// TIA Portal V16 export
// export: Created 2025-05-24T14:53:42.6954034Z, ExportSetting WithDefaults, DisplayName Totally Integrated Automation Portal, DisplayVersion V16, DisplayName TIA Portal Version Control Interface, DisplayVersion V16, DisplayName TIA Portal Openness, DisplayVersion V16, DisplayName STEP 7 Professional, DisplayVersion V16, DisplayName STEP 7 Safety, DisplayVersion V16, DisplayName WinCC Advanced, DisplayVersion V16
ORGANIZATION_BLOCK "OB1"   // OB1, LAD, ProgramCycle
TITLE = MAIN Program
VERSION : 0.1
// MAIN Block
// stored: IsIECCheckEnabled false
   VAR_TEMP
      Temp_0 : Byte;
      Temp_1 : Byte;
      Temp_2 : Byte;
      Temp_3 : Byte;
      Temp_4 : Byte;
      Temp_5 : Byte;
      Temp_6 : Int;
      Temp_7 : Int;
      Temp_8 : Int;
      Temp_9 : Date_And_Time;
      Temp_10 : DWord;
      EncoderDirection : Bool;
      HomingActive : Bool;
      EncError : Bool;
      SafetyActive : Bool;
      "Spare Drive 6" : Bool;
      "Spare Drive 7" : Bool;
      "Spare Drive 8" : Bool;
      "Spare Drive 9" : Bool;
      "Spare Drive 10" : Bool;
      SAFE_OK_Signal : Bool;
      Raw_Position : Real;
      Encoder : Int;
      Gate : Bool;
      GATESTP : Bool;
      OTERRA : Bool;
      Direct : Bool;
      Prepar : Bool;
      CMPV1 : Bool;
      CMPV2 : Bool;
      RESSYNC : Bool;
      RESZERO : Bool;
      OTERR : Bool;
      UnscPos : Int;
      Sc_Pos : Int;
      ActEncPos : Real;
      Start_ReferenceRun : Bool;
      ReferenceSwitch_Input : Bool;
      "Reference Position" : Real;
      "Jog FWD" : Bool;
      "Jog REV" : Bool;
      RefSwitchTemp : Bool;
      RefPosDint : DInt;
      RefPosInt : Real;
      Start_Movement : Bool;
      ClockTime : Int;
      LT_Time : Date_And_Time;
      Summer : Bool;
      SystemStartUp : Bool;
      StartupLow : Bool;
      ManualSensorOverride : Bool;
      Axis1_ScaledPosition : Real;
      Axis1_ActualEncPosition : Real;
   END_VAR
   VAR_TEMP   // added for the SCL form of the ladder/FBD networks
      _w1 : Bool;
   END_VAR
BEGIN

REGION Network 1: Retain Variables
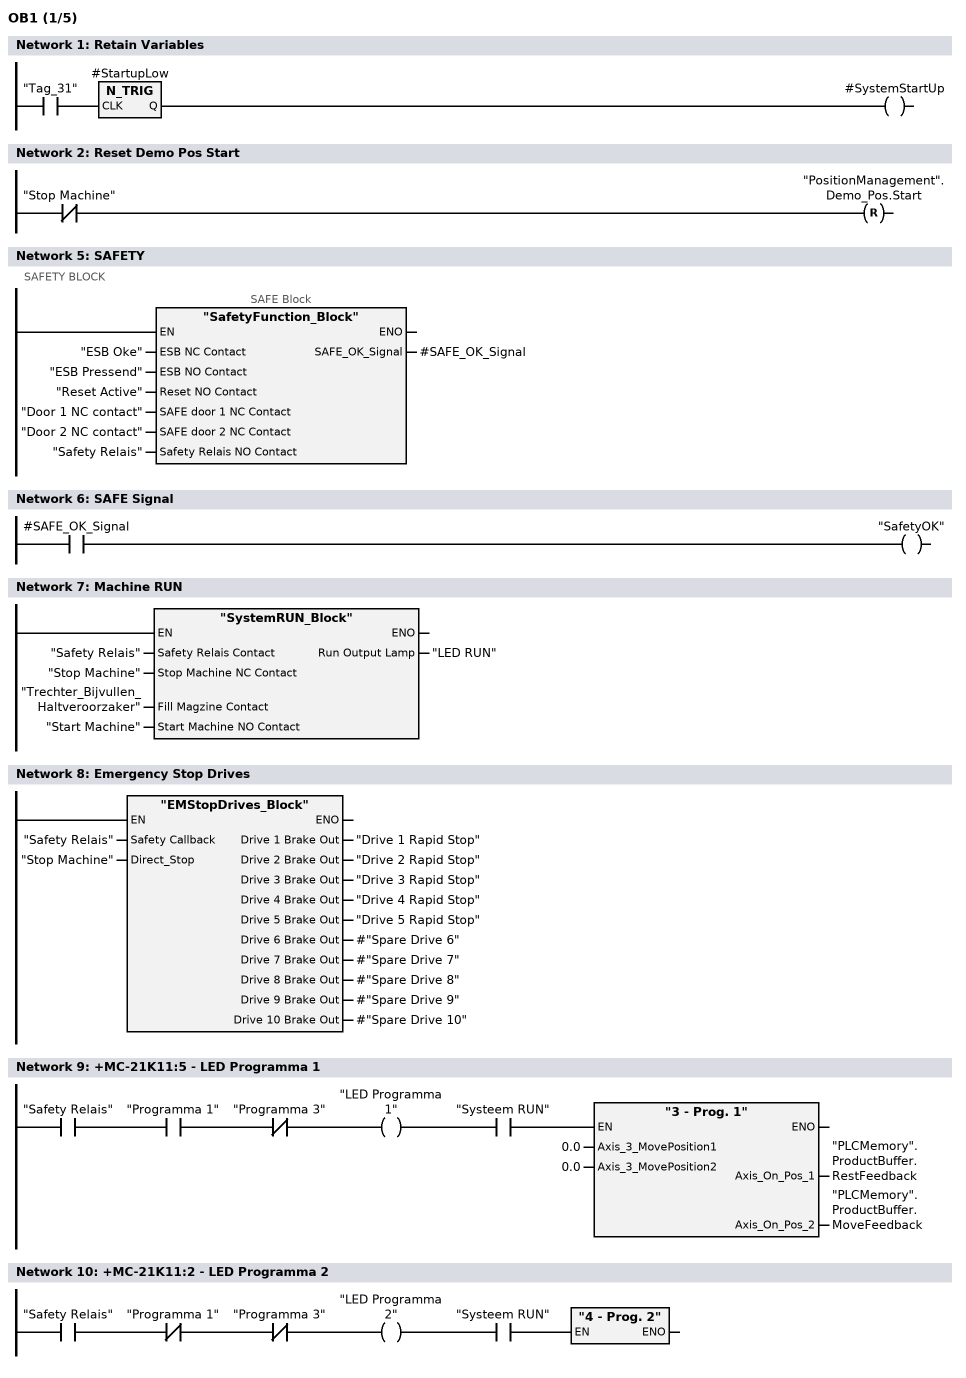
   RUNG wire#powerrail
      Contact( "Tag_31" )
      N_Trig( #StartupLow )
      Coil( #SystemStartUp )
   END_RUNG
   // the same network as SCL:
   #_w1 := NOT "Tag_31" AND #StartupLow;   // falling edge
   #StartupLow := "Tag_31";
   #SystemStartUp := #_w1;
END_REGION

REGION Network 2: Reset Demo Pos Start
   RUNG wire#powerrail
      I_Contact( "Stop Machine" )
      R_Coil( "PositionManagement".Demo_Pos.Start )
   END_RUNG
   // the same network as SCL:
   IF NOT "Stop Machine" THEN "PositionManagement".Demo_Pos.Start := FALSE; END_IF;
END_REGION

REGION Network 3: Retain Veriables (2)
END_REGION

REGION Network 4: System Time
END_REGION

REGION Network 5: SAFETY
   // SAFETY BLOCK
   RUNG wire#powerrail
      "SafetyFunction_Block"("ESB NC Contact" := "ESB Oke", "ESB NO Contact" := "ESB Pressend", "Reset NO Contact" := "Reset Active", "SAFE door 1 NC Contact" := "Door 1 NC contact", "SAFE door 2 NC Contact" := "Door 2 NC contact", "Safety Relais NO Contact" := "Safety Relais", SAFE_OK_Signal => #SAFE_OK_Signal)   // SAFE Block
   END_RUNG
   // the same network as SCL:
   "SafetyFunction_Block"("ESB NC Contact" := "ESB Oke",   // SAFE Block
                          "ESB NO Contact" := "ESB Pressend",
                          "Reset NO Contact" := "Reset Active",
                          "SAFE door 1 NC Contact" := "Door 1 NC contact",
                          "SAFE door 2 NC Contact" := "Door 2 NC contact",
                          "Safety Relais NO Contact" := "Safety Relais",
                          SAFE_OK_Signal => #SAFE_OK_Signal);
END_REGION

REGION Network 6: SAFE Signal
   RUNG wire#powerrail
      Contact( #SAFE_OK_Signal )
      Coil( "SafetyOK" )
   END_RUNG
   // the same network as SCL:
   "SafetyOK" := #SAFE_OK_Signal;
END_REGION

REGION Network 7: Machine RUN
   RUNG wire#powerrail
      "SystemRUN_Block"("Safety Relais Contact" := "Safety Relais", "Stop Machine NC Contact" := "Stop Machine", "Fill Magzine Contact" := "Trechter_Bijvullen_Haltveroorzaker", "Start Machine NO Contact" := "Start Machine", "Run Output Lamp" => "LED RUN")
   END_RUNG
   // the same network as SCL:
   "SystemRUN_Block"("Safety Relais Contact" := "Safety Relais",
                     "Stop Machine NC Contact" := "Stop Machine",
                     "Fill Magzine Contact" := "Trechter_Bijvullen_Haltveroorzaker",
                     "Start Machine NO Contact" := "Start Machine",
                     "Run Output Lamp" => "LED RUN");
END_REGION

REGION Network 8: Emergency Stop Drives
   RUNG wire#powerrail
      "EMStopDrives_Block"("Safety Callback" := "Safety Relais", Direct_Stop := "Stop Machine", "Drive 1 Brake Out" => "Drive 1 Rapid Stop", "Drive 2 Brake Out" => "Drive 2 Rapid Stop", "Drive 3 Brake Out" => "Drive 3 Rapid Stop", "Drive 4 Brake Out" => "Drive 4 Rapid Stop", "Drive 5 Brake Out" => "Drive 5 Rapid Stop", "Drive 6 Brake Out" => #"Spare Drive 6", "Drive 7 Brake Out" => #"Spare Drive 7", "Drive 8 Brake Out" => #"Spare Drive 8", "Drive 9 Brake Out" => #"Spare Drive 9", "Drive 10 Brake Out" => #"Spare Drive 10")
   END_RUNG
   // the same network as SCL:
   "EMStopDrives_Block"("Safety Callback" := "Safety Relais",
                        Direct_Stop := "Stop Machine",
                        "Drive 1 Brake Out" => "Drive 1 Rapid Stop",
                        "Drive 2 Brake Out" => "Drive 2 Rapid Stop",
                        "Drive 3 Brake Out" => "Drive 3 Rapid Stop",
                        "Drive 4 Brake Out" => "Drive 4 Rapid Stop",
                        "Drive 5 Brake Out" => "Drive 5 Rapid Stop",
                        "Drive 6 Brake Out" => #"Spare Drive 6",
                        "Drive 7 Brake Out" => #"Spare Drive 7",
                        "Drive 8 Brake Out" => #"Spare Drive 8",
                        "Drive 9 Brake Out" => #"Spare Drive 9",
                        "Drive 10 Brake Out" => #"Spare Drive 10");
END_REGION

REGION Network 9: +MC-21K11:5 - LED Programma 1
   RUNG wire#powerrail
      Contact( "Safety Relais" )
      Contact( "Programma 1" )
      I_Contact( "Programma 3" )
      Coil( "LED Programma 1" )
      Contact( "Systeem RUN" )
      "3 - Prog. 1"(Axis_3_MovePosition1 := 0.0, Axis_3_MovePosition2 := 0.0, Axis_On_Pos_1 => "PLCMemory".ProductBuffer.RestFeedback, Axis_On_Pos_2 => "PLCMemory".ProductBuffer.MoveFeedback)
   END_RUNG
   // the same network as SCL:
   "LED Programma 1" := "Safety Relais" AND "Programma 1" AND NOT "Programma 3";
   IF "LED Programma 1" AND "Systeem RUN" THEN
       "3 - Prog. 1"(Axis_3_MovePosition1 := 0.0,
                     Axis_3_MovePosition2 := 0.0,
                     Axis_On_Pos_1 => "PLCMemory".ProductBuffer.RestFeedback,
                     Axis_On_Pos_2 => "PLCMemory".ProductBuffer.MoveFeedback);
   END_IF;
END_REGION

REGION Network 10: +MC-21K11:2 - LED Programma 2
   RUNG wire#powerrail
      Contact( "Safety Relais" )
      I_Contact( "Programma 1" )
      I_Contact( "Programma 3" )
      Coil( "LED Programma 2" )
      Contact( "Systeem RUN" )
      "4 - Prog. 2"()
   END_RUNG
   // the same network as SCL:
   "LED Programma 2" := "Safety Relais" AND NOT "Programma 1" AND NOT "Programma 3";
   IF "LED Programma 2" AND "Systeem RUN" THEN "4 - Prog. 2"(); END_IF;
END_REGION

REGION Network 11: +MC-21K11:6 - LED Programma 3
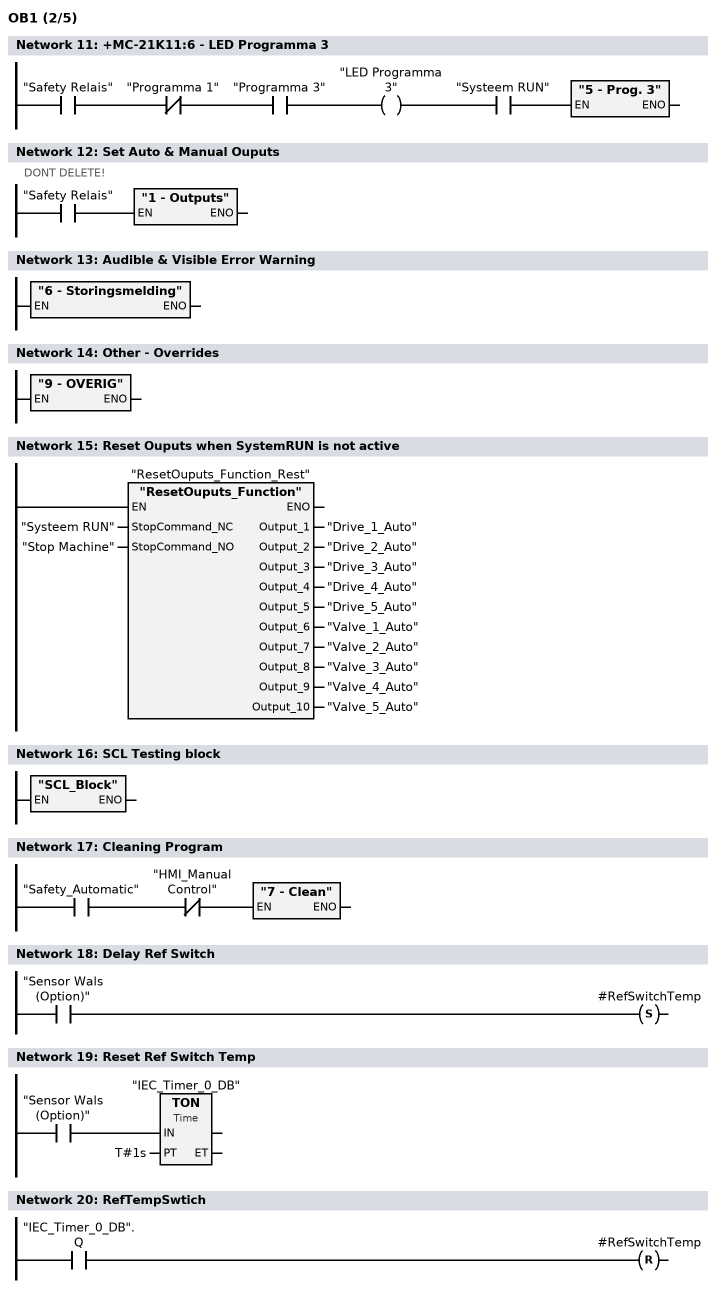
   RUNG wire#powerrail
      Contact( "Safety Relais" )
      I_Contact( "Programma 1" )
      Contact( "Programma 3" )
      Coil( "LED Programma 3" )
      Contact( "Systeem RUN" )
      "5 - Prog. 3"()
   END_RUNG
   // the same network as SCL:
   "LED Programma 3" := "Safety Relais" AND NOT "Programma 1" AND "Programma 3";
   IF "LED Programma 3" AND "Systeem RUN" THEN "5 - Prog. 3"(); END_IF;
END_REGION

REGION Network 12: Set Auto & Manual Ouputs
   // DONT DELETE!
   RUNG wire#powerrail
      Contact( "Safety Relais" )
      "1 - Outputs"()
   END_RUNG
   // the same network as SCL:
   IF "Safety Relais" THEN "1 - Outputs"(); END_IF;
END_REGION

REGION Network 13: Audible & Visible Error Warning
   RUNG wire#powerrail
      "6 - Storingsmelding"()
   END_RUNG
   // the same network as SCL:
   "6 - Storingsmelding"();
END_REGION

REGION Network 14: Other - Overrides
   RUNG wire#powerrail
      "9 - OVERIG"()
   END_RUNG
   // the same network as SCL:
   "9 - OVERIG"();
END_REGION

REGION Network 15: Reset Ouputs when SystemRUN is not active
   RUNG wire#powerrail
      "ResetOuputs_Function_Rest"(StopCommand_NC := "Systeem RUN", StopCommand_NO := "Stop Machine", Output_1 => "Drive_1_Auto", Output_2 => "Drive_2_Auto", Output_3 => "Drive_3_Auto", Output_4 => "Drive_4_Auto", Output_5 => "Drive_5_Auto", Output_6 => "Valve_1_Auto", Output_7 => "Valve_2_Auto", Output_8 => "Valve_3_Auto", Output_9 => "Valve_4_Auto", Output_10 => "Valve_5_Auto")
   END_RUNG
   // the same network as SCL:
   "ResetOuputs_Function_Rest"(StopCommand_NC := "Systeem RUN",   // "ResetOuputs_Function"
                           StopCommand_NO := "Stop Machine",
                           Output_1 => "Drive_1_Auto",
                           Output_2 => "Drive_2_Auto",
                           Output_3 => "Drive_3_Auto",
                           Output_4 => "Drive_4_Auto",
                           Output_5 => "Drive_5_Auto",
                           Output_6 => "Valve_1_Auto",
                           Output_7 => "Valve_2_Auto",
                           Output_8 => "Valve_3_Auto",
                           Output_9 => "Valve_4_Auto",
                           Output_10 => "Valve_5_Auto");
END_REGION

REGION Network 16: SCL Testing block
   RUNG wire#powerrail
      "SCL_Block"()
   END_RUNG
   // the same network as SCL:
   "SCL_Block"();
END_REGION

REGION Network 17: Cleaning Program
   RUNG wire#powerrail
      Contact( "Safety_Automatic" )
      I_Contact( "HMI_ManualControl" )
      "7 - Clean"()
   END_RUNG
   // the same network as SCL:
   IF "Safety_Automatic" AND NOT "HMI_ManualControl" THEN "7 - Clean"(); END_IF;
END_REGION

REGION Network 18: Delay Ref Switch
   RUNG wire#powerrail
      Contact( "Sensor Wals (Option)" )
      S_Coil( #RefSwitchTemp )
   END_RUNG
   // the same network as SCL:
   IF "Sensor Wals (Option)" THEN #RefSwitchTemp := TRUE; END_IF;
END_REGION

REGION Network 19: Reset Ref Switch Temp
   RUNG wire#powerrail
      Contact( "Sensor Wals (Option)" )
      { S7_Templates := "time_type := Time" } "IEC_Timer_0_DB".TON(pt := T#1s, et =>)
   END_RUNG
   // the same network as SCL:
   "IEC_Timer_0_DB".TON(IN := "Sensor Wals (Option)", PT := T#1s);
END_REGION

REGION Network 20: RefTempSwtich
   RUNG wire#powerrail
      Contact( "IEC_Timer_0_DB".Q )
      R_Coil( #RefSwitchTemp )
   END_RUNG
   // the same network as SCL:
   IF "IEC_Timer_0_DB".Q THEN #RefSwitchTemp := FALSE; END_IF;
END_REGION

REGION Network 21: Drive Manager Axis 3
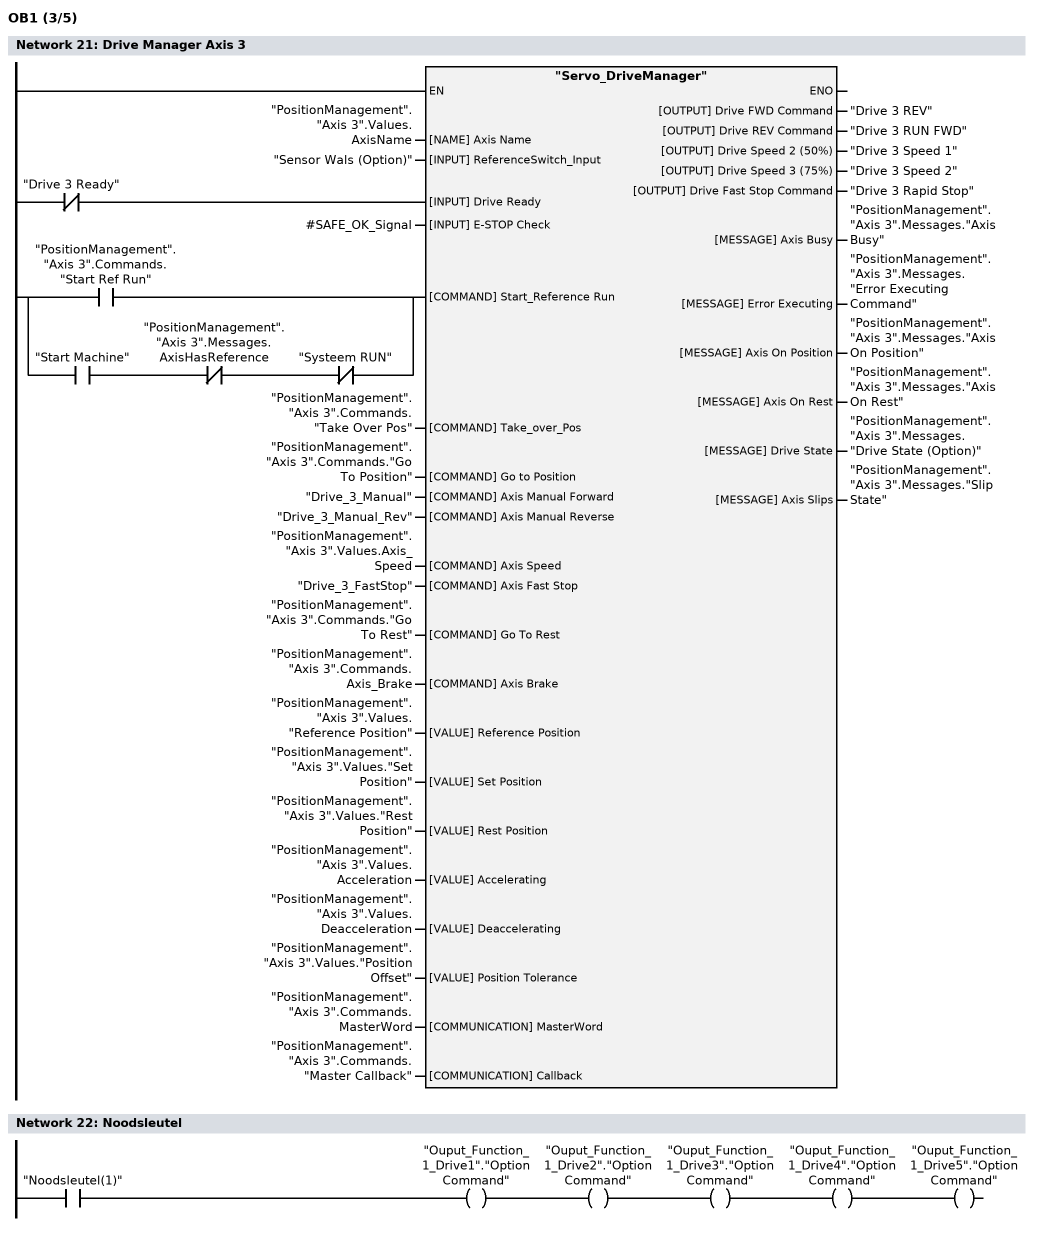
   RUNG wire#powerrail
      "Servo_DriveManager"("[INPUT] Drive Ready" := wire#w1, "[COMMAND] Start_Reference Run" := wire#w2, "[NAME] Axis Name" := "PositionManagement"."Axis 3".Values.AxisName, "[INPUT] ReferenceSwitch_Input" := "Sensor Wals (Option)", "[INPUT] E-STOP Check" := #SAFE_OK_Signal, "[COMMAND] Take_over_Pos" := "PositionManagement"."Axis 3".Commands."Take Over Pos", "[COMMAND] Go to Position" := "PositionManagement"."Axis 3".Commands."Go To Position", "[COMMAND] Axis Manual Forward" := "Drive_3_Manual", "[COMMAND] Axis Manual Reverse" := "Drive_3_Manual_Rev", "[COMMAND] Axis Speed" := "PositionManagement"."Axis 3".Values.Axis_Speed, "[COMMAND] Axis Fast Stop" := "Drive_3_FastStop", "[COMMAND] Go To Rest" := "PositionManagement"."Axis 3".Commands."Go To Rest", "[COMMAND] Axis Brake" := "PositionManagement"."Axis 3".Commands.Axis_Brake, "[VALUE] Reference Position" := "PositionManagement"."Axis 3".Values."Reference Position", "[VALUE] Set Position" := "PositionManagement"."Axis 3".Values."Set Position", "[VALUE] Rest Position" := "PositionManagement"."Axis 3".Values."Rest Position", "[VALUE] Accelerating" := "PositionManagement"."Axis 3".Values.Acceleration, "[VALUE] Deaccelerating" := "PositionManagement"."Axis 3".Values.Deacceleration, "[VALUE] Position Tolerance" := "PositionManagement"."Axis 3".Values."Position Offset", "[COMMUNICATION] MasterWord" := "PositionManagement"."Axis 3".Commands.MasterWord, "[COMMUNICATION] Callback" := "PositionManagement"."Axis 3".Commands."Master Callback", "[OUTPUT] Drive FWD Command" => "Drive 3 REV", "[OUTPUT] Drive REV Command" => "Drive 3 RUN FWD", "[OUTPUT] Drive Speed 2 (50%)" => "Drive 3 Speed 1", "[OUTPUT] Drive Speed 3 (75%)" => "Drive 3 Speed 2", "[OUTPUT] Drive Fast Stop Command" => "Drive 3 Rapid Stop", "[MESSAGE] Axis Busy" => "PositionManagement"."Axis 3".Messages."Axis Busy", "[MESSAGE] Error Executing" => "PositionManagement"."Axis 3".Messages."Error Executing Command", "[MESSAGE] Axis On Position" => "PositionManagement"."Axis 3".Messages."Axis On Position", "[MESSAGE] Axis On Rest" => "PositionManagement"."Axis 3".Messages."Axis On Rest", "[MESSAGE] Drive State" => "PositionManagement"."Axis 3".Messages."Drive State (Option)", "[MESSAGE] Axis Slips" => "PositionManagement"."Axis 3".Messages."Slip State")
   END_RUNG
   RUNG wire#powerrail
      I_Contact( "Drive 3 Ready" )
   END_RUNG wire#w1
   RUNG wire#powerrail
      Contact( "PositionManagement"."Axis 3".Commands."Start Ref Run" )
   END_RUNG wire#w2
   RUNG wire#powerrail
      Contact( "Start Machine" )
      I_Contact( "PositionManagement"."Axis 3".Messages.AxisHasReference )
      I_Contact( "Systeem RUN" )
   END_RUNG wire#w2
   // the same network as SCL:
   "Servo_DriveManager"("[NAME] Axis Name" := "PositionManagement"."Axis 3".Values.AxisName,
                        "[INPUT] ReferenceSwitch_Input" := "Sensor Wals (Option)",
                        "[INPUT] Drive Ready" := NOT "Drive 3 Ready",
                        "[INPUT] E-STOP Check" := #SAFE_OK_Signal,
                        "[COMMAND] Start_Reference Run" := "PositionManagement"."Axis 3".Commands."Start Ref Run" OR ("Start Machine" AND NOT "PositionManagement"."Axis 3".Messages.AxisHasReference AND NOT "Systeem RUN"),
                        "[COMMAND] Take_over_Pos" := "PositionManagement"."Axis 3".Commands."Take Over Pos",
                        "[COMMAND] Go to Position" := "PositionManagement"."Axis 3".Commands."Go To Position",
                        "[COMMAND] Axis Manual Forward" := "Drive_3_Manual",
                        "[COMMAND] Axis Manual Reverse" := "Drive_3_Manual_Rev",
                        "[COMMAND] Axis Speed" := "PositionManagement"."Axis 3".Values.Axis_Speed,
                        "[COMMAND] Axis Fast Stop" := "Drive_3_FastStop",
                        "[COMMAND] Go To Rest" := "PositionManagement"."Axis 3".Commands."Go To Rest",
                        "[COMMAND] Axis Brake" := "PositionManagement"."Axis 3".Commands.Axis_Brake,
                        "[VALUE] Reference Position" := "PositionManagement"."Axis 3".Values."Reference Position",
                        "[VALUE] Set Position" := "PositionManagement"."Axis 3".Values."Set Position",
                        "[VALUE] Rest Position" := "PositionManagement"."Axis 3".Values."Rest Position",
                        "[VALUE] Accelerating" := "PositionManagement"."Axis 3".Values.Acceleration,
                        "[VALUE] Deaccelerating" := "PositionManagement"."Axis 3".Values.Deacceleration,
                        "[VALUE] Position Tolerance" := "PositionManagement"."Axis 3".Values."Position Offset",
                        "[COMMUNICATION] MasterWord" := "PositionManagement"."Axis 3".Commands.MasterWord,
                        "[COMMUNICATION] Callback" := "PositionManagement"."Axis 3".Commands."Master Callback",
                        "[OUTPUT] Drive FWD Command" => "Drive 3 REV",
                        "[OUTPUT] Drive REV Command" => "Drive 3 RUN FWD",
                        "[OUTPUT] Drive Speed 2 (50%)" => "Drive 3 Speed 1",
                        "[OUTPUT] Drive Speed 3 (75%)" => "Drive 3 Speed 2",
                        "[OUTPUT] Drive Fast Stop Command" => "Drive 3 Rapid Stop",
                        "[MESSAGE] Axis Busy" => "PositionManagement"."Axis 3".Messages."Axis Busy",
                        "[MESSAGE] Error Executing" => "PositionManagement"."Axis 3".Messages."Error Executing Command",
                        "[MESSAGE] Axis On Position" => "PositionManagement"."Axis 3".Messages."Axis On Position",
                        "[MESSAGE] Axis On Rest" => "PositionManagement"."Axis 3".Messages."Axis On Rest",
                        "[MESSAGE] Drive State" => "PositionManagement"."Axis 3".Messages."Drive State (Option)",
                        "[MESSAGE] Axis Slips" => "PositionManagement"."Axis 3".Messages."Slip State");
END_REGION

REGION Network 22: Noodsleutel
   RUNG wire#powerrail
      Contact( "Noodsleutel(1)" )
      Coil( "Ouput_Function_1_Drive1"."Option Command" )
      Coil( "Ouput_Function_1_Drive2"."Option Command" )
      Coil( "Ouput_Function_1_Drive3"."Option Command" )
      Coil( "Ouput_Function_1_Drive4"."Option Command" )
      Coil( "Ouput_Function_1_Drive5"."Option Command" )
   END_RUNG
   // the same network as SCL:
   "Ouput_Function_1_Drive1"."Option Command" := "Noodsleutel(1)";
   "Ouput_Function_1_Drive2"."Option Command" := "Noodsleutel(1)";
   "Ouput_Function_1_Drive3"."Option Command" := "Noodsleutel(1)";
   "Ouput_Function_1_Drive4"."Option Command" := "Noodsleutel(1)";
   "Ouput_Function_1_Drive5"."Option Command" := "Noodsleutel(1)";
END_REGION

REGION Network 23: MC_Move (Manual)
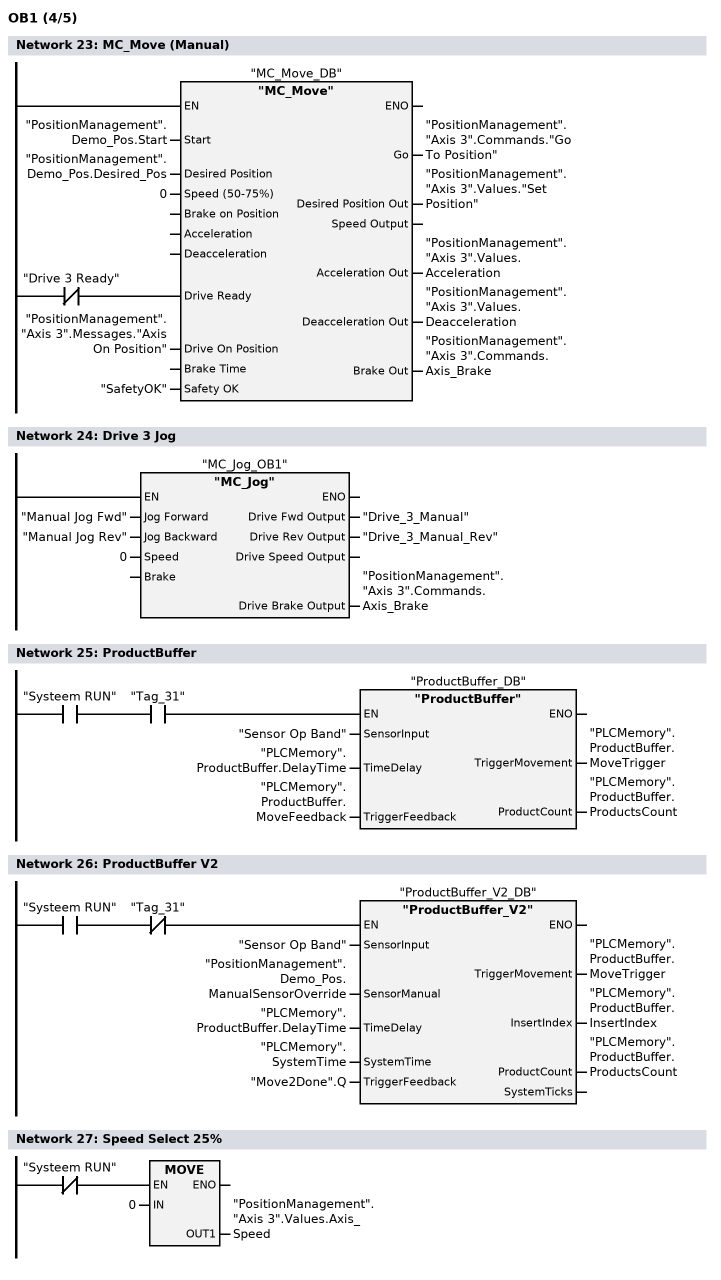
   RUNG wire#powerrail
      "MC_Move_DB"("Drive Ready" := wire#w1, Start := "PositionManagement".Demo_Pos.Start, "Desired Position" := "PositionManagement".Demo_Pos.Desired_Pos, "Speed (50-75%)" := 0, "Brake on Position" :=, Acceleration :=, Deacceleration :=, "Drive On Position" := "PositionManagement"."Axis 3".Messages."Axis On Position", "Brake Time" :=, "Safety OK" := "SafetyOK", Go => "PositionManagement"."Axis 3".Commands."Go To Position", "Desired Position Out" => "PositionManagement"."Axis 3".Values."Set Position", "Speed Output" =>, "Acceleration Out" => "PositionManagement"."Axis 3".Values.Acceleration, "Deacceleration Out" => "PositionManagement"."Axis 3".Values.Deacceleration, "Brake Out" => "PositionManagement"."Axis 3".Commands.Axis_Brake)
   END_RUNG
   RUNG wire#powerrail
      I_Contact( "Drive 3 Ready" )
   END_RUNG wire#w1
   // the same network as SCL:
   "MC_Move_DB"(Start := "PositionManagement".Demo_Pos.Start,   // "MC_Move"
                "Desired Position" := "PositionManagement".Demo_Pos.Desired_Pos,
                "Speed (50-75%)" := 0,
                "Drive Ready" := NOT "Drive 3 Ready",
                "Drive On Position" := "PositionManagement"."Axis 3".Messages."Axis On Position",
                "Safety OK" := "SafetyOK",
                Go => "PositionManagement"."Axis 3".Commands."Go To Position",
                "Desired Position Out" => "PositionManagement"."Axis 3".Values."Set Position",
                "Acceleration Out" => "PositionManagement"."Axis 3".Values.Acceleration,
                "Deacceleration Out" => "PositionManagement"."Axis 3".Values.Deacceleration,
                "Brake Out" => "PositionManagement"."Axis 3".Commands.Axis_Brake);
END_REGION

REGION Network 24: Drive 3 Jog
   RUNG wire#powerrail
      "MC_Jog_OB1"("Jog Forward" := "Manual Jog Fwd", "Jog Backward" := "Manual Jog Rev", Speed := 0, Brake :=, "Drive Fwd Output" => "Drive_3_Manual", "Drive Rev Output" => "Drive_3_Manual_Rev", "Drive Speed Output" =>, "Drive Brake Output" => "PositionManagement"."Axis 3".Commands.Axis_Brake)
   END_RUNG
   // the same network as SCL:
   "MC_Jog_OB1"("Jog Forward" := "Manual Jog Fwd",   // "MC_Jog"
                "Jog Backward" := "Manual Jog Rev",
                Speed := 0,
                "Drive Fwd Output" => "Drive_3_Manual",
                "Drive Rev Output" => "Drive_3_Manual_Rev",
                "Drive Brake Output" => "PositionManagement"."Axis 3".Commands.Axis_Brake);
END_REGION

REGION Network 25: ProductBuffer
   RUNG wire#powerrail
      Contact( "Systeem RUN" )
      Contact( "Tag_31" )
      "ProductBuffer_DB"(SensorInput := "Sensor Op Band", TimeDelay := "PLCMemory".ProductBuffer.DelayTime, TriggerFeedback := "PLCMemory".ProductBuffer.MoveFeedback, TriggerMovement => "PLCMemory".ProductBuffer.MoveTrigger, ProductCount => "PLCMemory".ProductBuffer.ProductsCount)
   END_RUNG
   // the same network as SCL:
   IF "Systeem RUN" AND "Tag_31" THEN
       "ProductBuffer_DB"(SensorInput := "Sensor Op Band",   // "ProductBuffer"
                          TimeDelay := "PLCMemory".ProductBuffer.DelayTime,
                          TriggerFeedback := "PLCMemory".ProductBuffer.MoveFeedback,
                          TriggerMovement => "PLCMemory".ProductBuffer.MoveTrigger,
                          ProductCount => "PLCMemory".ProductBuffer.ProductsCount);
   END_IF;
END_REGION

REGION Network 26: ProductBuffer V2
   RUNG wire#powerrail
      Contact( "Systeem RUN" )
      I_Contact( "Tag_31" )
      "ProductBuffer_V2_DB"(SensorInput := "Sensor Op Band", SensorManual := "PositionManagement".Demo_Pos.ManualSensorOverride, TimeDelay := "PLCMemory".ProductBuffer.DelayTime, SystemTime := "PLCMemory".SystemTime, TriggerFeedback := "Move2Done".Q, TriggerMovement => "PLCMemory".ProductBuffer.MoveTrigger, InsertIndex => "PLCMemory".ProductBuffer.InsertIndex, ProductCount => "PLCMemory".ProductBuffer.ProductsCount, SystemTicks =>)
   END_RUNG
   // the same network as SCL:
   IF "Systeem RUN" AND NOT "Tag_31" THEN
       "ProductBuffer_V2_DB"(SensorInput := "Sensor Op Band",   // "ProductBuffer_V2"
                             SensorManual := "PositionManagement".Demo_Pos.ManualSensorOverride,
                             TimeDelay := "PLCMemory".ProductBuffer.DelayTime,
                             SystemTime := "PLCMemory".SystemTime,
                             TriggerFeedback := "Move2Done".Q,
                             TriggerMovement => "PLCMemory".ProductBuffer.MoveTrigger,
                             InsertIndex => "PLCMemory".ProductBuffer.InsertIndex,
                             ProductCount => "PLCMemory".ProductBuffer.ProductsCount);
   END_IF;
END_REGION

REGION Network 27: Speed Select 25%
   RUNG wire#powerrail
      I_Contact( "Systeem RUN" )
      { S7_GenerateENO := "TRUE" } Move(in := 0, out1 => "PositionManagement"."Axis 3".Values.Axis_Speed)
   END_RUNG
   // the same network as SCL:
   IF NOT "Systeem RUN" THEN "PositionManagement"."Axis 3".Values.Axis_Speed := 0; END_IF;
END_REGION

REGION Network 28: Speed Select 75%
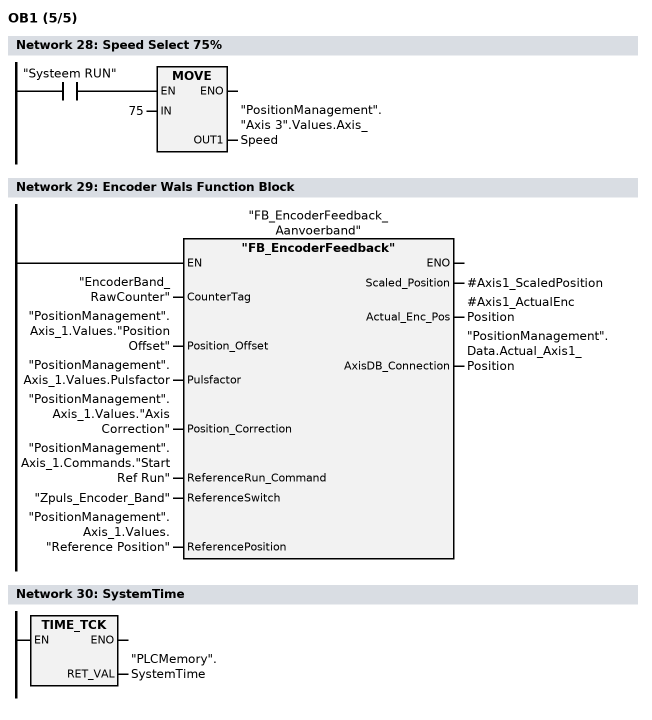
   RUNG wire#powerrail
      Contact( "Systeem RUN" )
      { S7_GenerateENO := "TRUE" } Move(in := 75, out1 => "PositionManagement"."Axis 3".Values.Axis_Speed)
   END_RUNG
   // the same network as SCL:
   IF "Systeem RUN" THEN "PositionManagement"."Axis 3".Values.Axis_Speed := 75; END_IF;
END_REGION

REGION Network 29: Encoder Wals Function Block
   RUNG wire#powerrail
      "FB_EncoderFeedback_Aanvoerband"(CounterTag := "EncoderBand_RawCounter", Position_Offset := "PositionManagement".Axis_1.Values."Position Offset", Pulsfactor := "PositionManagement".Axis_1.Values.Pulsfactor, Position_Correction := "PositionManagement".Axis_1.Values."Axis Correction", ReferenceRun_Command := "PositionManagement".Axis_1.Commands."Start Ref Run", ReferenceSwitch := "Zpuls_Encoder_Band", ReferencePosition := "PositionManagement".Axis_1.Values."Reference Position", Scaled_Position => #Axis1_ScaledPosition, Actual_Enc_Pos => #Axis1_ActualEncPosition, AxisDB_Connection => "PositionManagement".Data.Actual_Axis1_Position)
   END_RUNG
   // the same network as SCL:
   "FB_EncoderFeedback_Aanvoerband"(CounterTag := "EncoderBand_RawCounter",   // "FB_EncoderFeedback"
                           Position_Offset := "PositionManagement".Axis_1.Values."Position Offset",
                           Pulsfactor := "PositionManagement".Axis_1.Values.Pulsfactor,
                           Position_Correction := "PositionManagement".Axis_1.Values."Axis Correction",
                           ReferenceRun_Command := "PositionManagement".Axis_1.Commands."Start Ref Run",
                           ReferenceSwitch := "Zpuls_Encoder_Band",
                           ReferencePosition := "PositionManagement".Axis_1.Values."Reference Position",
                           Scaled_Position => #Axis1_ScaledPosition,
                           Actual_Enc_Pos => #Axis1_ActualEncPosition,
                           AxisDB_Connection => "PositionManagement".Data.Actual_Axis1_Position);
END_REGION

REGION Network 30: SystemTime
   RUNG wire#powerrail
      TIME_TCK(RET_VAL => "PLCMemory".SystemTime)
   END_RUNG
   // the same network as SCL:
   "PLCMemory".SystemTime := TIME_TCK();
END_REGION
END_ORGANIZATION_BLOCK
